Staubli VAL3: removeTraj.pgx

public program removeTraj()
begin
  // mutex it
  setMutex(bActionMutex)
  if saveData:bDebug
    ? "CYCLESTATUS: TRAJ Remove "+tTrajCycle.sID
  endIf
  // remove the action
  if size(tTrajCycle)>1
    delete(tTrajCycle[0])
  else
    // reset
    resize(tTrajCycle.tSuper,1,1)
    tTrajCycle.sID="null"
    tTrajCycle.nId=0
  endIf
  // release
  bActionMutex=false
end
